SUBAPPLICATION SwitchPic_2_3 (* Bild umschalten VT SK, AUX und VT Button; 2 Zustände *)
  (* Standard: 61499-2 *)
  (* Version 1.0, 2026-05-29, franz *)
  PACKAGE MyLib::sys;
  IMPORT isobus::UT::Q::const::IDs::ID_NULL;
  IMPORT isobus::UT::Q::types::s2x2ObjectIDs;
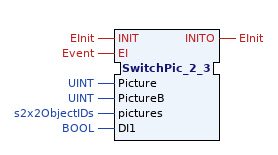
  EVENT_INPUT
    INIT : EInit; (* Initialization Request *)
    EI;
  END_EVENT
  EVENT_OUTPUT
    INITO : EInit; (* Initialization Confirm *)
  END_EVENT
  VAR_INPUT
    Picture : UINT; (* Object ID of the ObjectPointer to the Picture (SK) *)
    PictureB : UINT; (* Object ID of the ObjectPointer to the Picture (Button) *)
    pictures : isobus::UT::Q::types::s2x2ObjectIDs := (up := (u16ObjId := ID_NULL, u16ObjIdA := ID_NULL), down := (u16ObjId := ID_NULL, u16ObjIdA := ID_NULL)); (* the single Pictures *)
    DI1 : BOOL := FALSE; (* Selector *)
  END_VAR
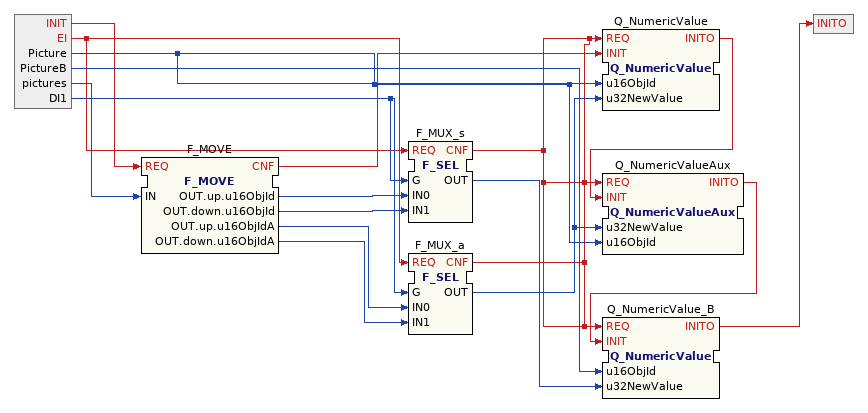
  FBS
    Q_NumericValue : isobus::UT::Q::Q_NumericValue;
    Q_NumericValueAux : isobus::UT::Q::Q_NumericValueAux;
    Q_NumericValue_B : isobus::UT::Q::Q_NumericValue;
    F_MOVE : iec61131::selection::F_MOVE; {SET_ATTRIBUTE(DataType, isobus::UT::Q::types::s2x2ObjectIDs)}
    F_MUX_s : iec61131::selection::F_SEL;
    F_MUX_a : iec61131::selection::F_SEL;
  END_FBS
  EVENT_CONNECTIONS
    EI TO F_MUX_s.REQ;
    F_MUX_s.CNF TO Q_NumericValue.REQ;
    F_MUX_s.CNF TO Q_NumericValueAux.REQ;
    F_MUX_s.CNF TO Q_NumericValue_B.REQ;
    INIT TO F_MOVE.REQ;
    F_MOVE.CNF TO Q_NumericValue.INIT;
    Q_NumericValue.INITO TO Q_NumericValueAux.INIT;
    Q_NumericValueAux.INITO TO Q_NumericValue_B.INIT;
    Q_NumericValue_B.INITO TO INITO;
    F_MUX_a.CNF TO Q_NumericValue.REQ;
    F_MUX_a.CNF TO Q_NumericValueAux.REQ;
    F_MUX_a.CNF TO Q_NumericValue_B.REQ;
    EI TO F_MUX_a.REQ;
  END_CONNECTIONS
  DATA_CONNECTIONS
    Picture TO Q_NumericValue.u16ObjId;
    PictureB TO Q_NumericValue_B.u16ObjId;
    pictures TO F_MOVE.IN;
    DI1 TO F_MUX_s.G;
    F_MUX_a.OUT TO Q_NumericValue.u32NewValue;
    F_MUX_a.OUT TO Q_NumericValueAux.u32NewValue;
    F_MOVE.OUT.up.u16ObjId TO F_MUX_s.IN0;
    F_MOVE.OUT.down.u16ObjId TO F_MUX_s.IN1;
    DI1 TO F_MUX_a.G;
    F_MOVE.OUT.up.u16ObjIdA TO F_MUX_a.IN0;
    F_MOVE.OUT.down.u16ObjIdA TO F_MUX_a.IN1;
    F_MUX_s.OUT TO Q_NumericValue_B.u32NewValue;
    Picture TO Q_NumericValueAux.u16ObjId;
  END_CONNECTIONS
END_SUBAPPLICATION
